// TwinCAT 3 PLC project Bsc_NoComp
// ProgramVersion: 3.1.4024.0
// libraries:
//   Tc2_Standard, * (Beckhoff Automation GmbH)
//   Tc2_System, * (Beckhoff Automation GmbH)
//   Tc3_Module, * (Beckhoff Automation GmbH)
// project tree:
//   GVLs/ G_Enables.TcGVL (not stored), G_FilterConstants.TcGVL (not stored), G_Mode.TcGVL (not stored), G_OPC.TcGVL (not stored), G_Parameters.TcGVL
//   Input/ G_Input.TcGVL
//   Output/ G_Output.TcGVL
//   / PlcTask.TcTTO
//   Program/ MAIN.TcPOU (not stored)
//   XML/ FB_Derivator.TcPOU (not stored), FB_Integrator.TcPOU (not stored), G_Init.TcGVL (not stored)
// real-time tasks:
//   TASK PlcTask: cycle T#1ms, priority 20, ADS port 350

CONFIGURATION Bsc_NoComp
    RESOURCE PLC ON TwinCAT3
        TASK PlcTask(INTERVAL := T#10ms, PRIORITY := 20);
        PROGRAM MAIN WITH PlcTask : MAIN;
    END_RESOURCE
END_CONFIGURATION

// ---- GVLs/G_Parameters.TcGVL
{attribute 'qualified_only'}
VAR_GLOBAL
END_VAR

// ---- Input/G_Input.TcGVL
{attribute 'qualified_only'}
VAR_GLOBAL
END_VAR

// ---- Output/G_Output.TcGVL
{attribute 'qualified_only'}
VAR_GLOBAL
END_VAR
